// TIA Portal V20 export
FUNCTION_BLOCK "FB_TimeCounter"   // FB53, SCL
{ S7_Optimized_Access := 'TRUE' }
// stored: MemoryReserve 100, SetENOAutomatically false
   VAR_INPUT
      iStart : Bool;
      iReset : Bool;
   END_VAR
   VAR_IN_OUT
      ioHours : Int;
      ioMinutes : Int;
      ioSeconds : Int;
      ioHoursCumul : Int;
      ioMinutesCumul : Int;
      ioSecondsCumul : DInt;
   END_VAR
   VAR
      sRT_Second { ExternalAccessible := 'False'; ExternalVisible := 'False'; ExternalWritable := 'False'} : R_TRIG;
   END_VAR
BEGIN
   REGION Description header 
       //==================================================================================
       // POSALUX Swiss SA / (C) Copyright 2025
       //----------------------------------------------------------------------------------
       // Title: Timer Counter
       // Comment/Function: This function allows:
       //                      - Counting Hours - Minutes - Seconds 
       //                      - Pulse each Hour - Minute - Second
       //
       // Author: Fabien Waldt
       // Engineering: TIA Portal v17
       //----------------------------------------------------------------------------------
       // Change log table:
       // Version  | Date     | Expert in charge | Changes applied
       // ---------|----------|------------------|------------------------------------
       // 00.00.01 | 20250314 | WFA              | First released version
       // ==================================================================================
   END_REGION

   //"Seconds" rising edge
   #sRT_Second(CLK := "Clock_1Hz");

   REGION Time counters reset
       IF #iReset THEN
           #ioHours := 0;
           #ioMinutes := 0;
           #ioSeconds := 0;
           #ioHoursCumul := 0;
           #ioMinutesCumul := 0;
           #ioSecondsCumul := 0;
       END_IF;
   END_REGION

   REGION Time counters
   IF #iStart AND #sRT_Second.Q THEN
       #ioSeconds := #ioSeconds + 1;
       #ioSecondsCumul := #ioSecondsCumul + 1;
       IF #ioSeconds >= 60 THEN
           #ioMinutes := #ioMinutes + 1;
           #ioSeconds := 0;
           #ioMinutesCumul := #ioMinutesCumul + 1;
           IF #ioMinutes >= 60 THEN
               #ioHours := #ioHours + 1;
               #ioMinutes := 0;
               #ioHoursCumul := #ioHoursCumul + 1;
           END_IF;
       END_IF;
   END_IF;
   END_REGION
END_FUNCTION_BLOCK
